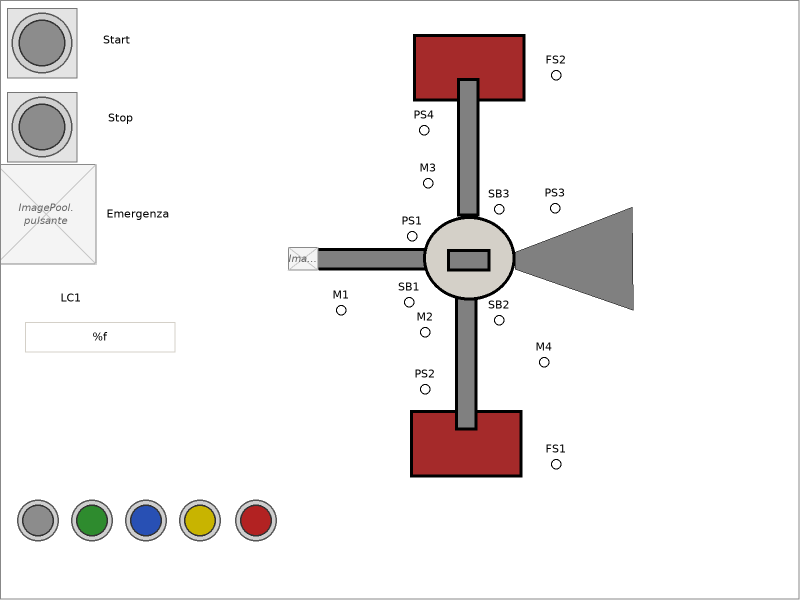
VISUALIZATION Visualization  // 800x600
    Rectangle (473,-103 67x112), angle 270
    Rectangle (470,273 67x112), angle 270
    PushSwitch (7,8 70x70), variable: GVL.PB1, behaviour: TAP, style: Switch-PushSwitch-Gray
    Label (89,25 55x30), "Start"
    PushSwitch (7,92 70x70), variable: GVL.PB2, behaviour: TAP, style: Switch-PushSwitch-Gray
    Label (88,103 65x30), "Stop"
    Label (93,199 90x30), "Emergenza"
    Rectangle (289,248 138x22)
    Rectangle (304,201 138x22), angle 90
    Rectangle (302,415 138x22), angle 90
    Ellipse (423,216 92x84)
    Polygon (515,252) (557,236) (632,207) (633,310) (515,269)
    Ellipse (407,231 10x10), colour toggle: GVL.PS1
        tap GVL.PS1
    Label (388,215 48x12), "PS1"
    Lamp1 (14,496 48x49), variable: GVL.L1, style: Lamp-Lamp1-Gray
    Lamp1 (68,496 48x49), variable: GVL.L2, style: Lamp-Lamp1-Green
    Lamp1 (122,496 48x49), variable: GVL.L3, style: Lamp-Lamp1-Blue
    Lamp1 (176,496 48x49), variable: GVL.L4, style: Lamp-Lamp1-Yellow
    Lamp1 (232,496 48x49), variable: GVL.L5, style: Lamp-Lamp1-Red
    Ellipse (551,459 10x10), colour toggle: GVL.FS1
        toggle GVL.FS1
    Label (532,443 48x12), "FS1"
    Ellipse (551,70 10x10), colour toggle: GVL.FS2
        toggle GVL.FS2
    Label (532,54 48x12), "FS2"
    Ellipse (420,384 10x10), colour toggle: GVL.PS2
        tap GVL.PS2
    Label (401,368 48x12), "PS2"
    Ellipse (550,203 10x10), colour toggle: GVL.PS3
        tap GVL.PS3
    Label (531,187 48x12), "PS3"
    Ellipse (419,125 10x10), colour toggle: GVL.PS4
        tap GVL.PS4
    Label (400,109 48x12), "PS4"
    Label (317,289 48x12), "M1"
    Ellipse (336,305 10x10), colour toggle: GVL.M1
    Label (401,311 48x12), "M2"
    Ellipse (420,327 10x10), colour toggle: GVL.M2
    Label (404,162 48x12), "M3"
    Ellipse (423,178 10x10), colour toggle: GVL.M3
    Label (520,341 48x12), "M4"
    Ellipse (539,357 10x10), colour toggle: GVL.M4
    Textfield (25,322 150x30), "%f", text variable: GVL.LC1
        OnMouseClick: write GVL.LC1 via VisuDialogs.Numpad, min 0, max 10
    Label (26,283 90x30), "LC1"
    Ellipse (494,315 10x10), colour toggle: GVL.SB2
        toggle GVL.SB2
    Label (475,299 48x12), "SB2"
    Label (475,188 48x12), "SB3"
    Ellipse (494,204 10x10), colour toggle: GVL.SB3
        toggle GVL.SB3
    Label (385,281 48x12), "SB1"
    Ellipse (404,297 10x10), colour toggle: GVL.SB1
        toggle GVL.SB1
    Rectangle (447,249 43x22), angle 180, colour toggle: GVL.M5
        p2858320360: VISU.rotazionePiattaforma
    Image (288,247 30x23), invisible if: NOT VISU.prosciuttoVisibile, image: ImagePool.ham
        p3560616238: VISU.posizioneProsciutto
        p2858320360: VISU.rotazionePiattaforma
        p2738717112: VISU.posizioneProsciuttoY
    Image (-4,164 100x100), image: ImagePool.pulsante
        OnMouseClick: toggle GVL.PBE
END_VISUALIZATION

(* stored: Version 1.1.0.1, ProductVersion 3.1.4024.12
   Visu Visualization: Id {e3399594-b7fd-4589-9a49-3967da9e8e84} *)
